// TIA Portal V19 export
DATA_BLOCK "DB_SNTP_Param"   // DB201
{ S7_Optimized_Access := 'TRUE' }
// stored: AutoNumber false, MemoryReserve 100
   VAR
      referenceID : USInt;   // Source of date and time (0 = uncalibrated local clock, 1 = DCF77, 2 = GPS)
      lastTimeSet : DTL := DTL#1990-01-01-00:00:00;   // Date and time when the time was set last. Set only if external reference is used.
      connID : CONN_OUC := 16#0FFF;   // Internal connection ID used for TURCV and TUSEND
   END_VAR
BEGIN
END_DATA_BLOCK
